# B&R Automation Studio project po_lab4
Automation Studio 4.5.2.102

## Configuration Real

### Hardware
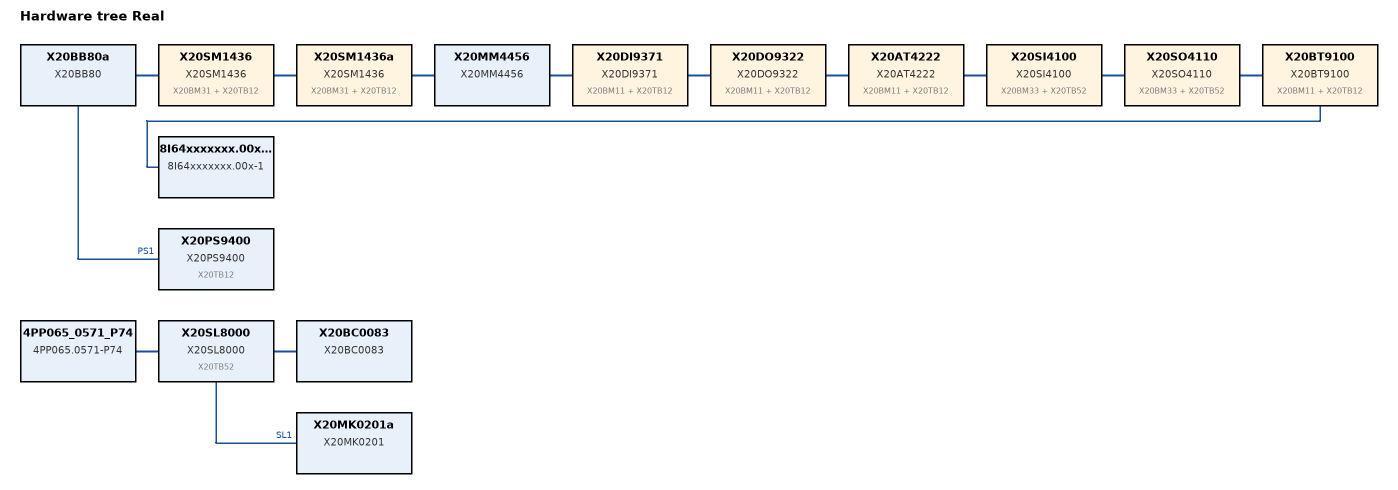
```
4PP065_0571_P74 : 4PP065.0571-P74 v1.1.2.0
  Connector IF4:
    EplInterfaceRedundant = 0
    EplEthInterfaceRedundant = 0
  Connector IF5:
    ActivateDevice = 1
    Mode = Manual
    InternetAddress = 10.0.1.10
    SubnetMask = 255.255.255.0
  ConfigurationID = LabBR
  TimerDeviceType = EPLX2X
  TimerDevice = 4PP065_0571_P74.IF4
  TaskClassIdleTime = 2000
  Cyclic1Tolerance = 0
  Cyclic1Output = 1
  Cyclic3Tolerance = 0
  VcObjectName = Visu
8I64xxxxxxx.00x-1 : 8I64xxxxxxx.00x-1 v1.3.9.1  [X2X1 -> X20BT9100.X2X1 [Cable Type=X2XCable, Length=10, Version=1.0.0.2]]
  BothEndSwitchesAreNormallyOpen_r1 = on
  QuickStopIsNormallyOpen_r1 = on
X20AT4222 : X20AT4222 v1.2.3.0  [SS1 -> X20TB12f.SS; SL -> X20BM11c.SL1]
X20BB80a : X20BB80 v1.0.2.0
X20BC0083 : X20BC0083 v2.7.0.0  [PLK1 -> X20SL8000.PLK2 (NodeNumber=2) [Cable Type=PowerlinkCable, Length=10, Version=1.0.0.2]; SL -> X20BB80a.SL1]
X20BM11a : X20BM11 v1.0.0.1  [X2X1 -> X20MM4456.X2X2]
X20BM11b : X20BM11 v1.0.0.1  [X2X1 -> X20BM11a.X2X2]
X20BM11c : X20BM11 v1.0.0.1  [X2X1 -> X20BM11b.X2X2]
X20BM11d : X20BM11 v1.0.0.1  [X2X1 -> X20BM33b.X2X2]
X20BM31a : X20BM31 v1.0.0.1  [X2X1 -> X20BB80a.IF1]
X20BM31b : X20BM31 v1.0.0.1  [X2X1 -> X20BM31a.X2X2]
X20BM33a : X20BM33 v1.0.0.4  [X2X1 -> X20BM11c.X2X2]
X20BM33b : X20BM33 v1.0.0.4  [X2X1 -> X20BM33a.X2X2]
X20BT9100 : X20BT9100 v1.0.3.0  [SS1 -> X20TB12g.SS; SL -> X20BM11d.SL1]
X20DI9371 : X20DI9371 v1.0.2.0  [SS1 -> X20TB12d.SS; SL -> X20BM11a.SL1]
X20DO9322 : X20DO9322 v1.0.3.0  [SS1 -> X20TB12e.SS; SL -> X20BM11b.SL1]
X20MK0201a : X20MK0201 v1.0.0.0  [SL -> X20SL8000.SL1]
X20MM4456 : X20MM4456 v1.1.5.0  [X2X1 -> X20BM31b.X2X2]
X20PS9400 : X20PS9400 v1.0.2.4  [SS1 -> X20TB12b.SS; PS -> X20BB80a.PS1]
X20SI4100 : X20SI4100 v1.10.1.1  [SS1 -> X20TB52b.SS; SL -> X20BM33a.SL1]
X20SL8000 : X20SL8000 v1.6.5.1  [PLK1 -> 4PP065_0571_P74.IF4 (NodeNumber=1) [Cable Type=PowerlinkCable, Length=10, Version=1.0.0.2]; PLK2 -> X20BC0083.PLK1 (NodeNumber=1) [Cable Type=PowerlinkCable, Length=10, Version=1.0.0.2]; SS1 -> X20TB52a.SS]
  SafeProject = SafeLOGIC-1
X20SM1436 : X20SM1436 v1.4.2.1  [SS1 -> X20TB12a.SS; SL -> X20BM31a.SL1]
X20SM1436a : X20SM1436 v1.4.2.1  [SS1 -> X20TB12c.SS; SL -> X20BM31b.SL1]
X20SO4110 : X20SO4110 v1.10.1.1  [SS1 -> X20TB52c.SS; SL -> X20BM33b.SL1]
  SafeLogicID = 2
  SafeModuleID = 3
X20TB12a : X20TB12 v1.0.0.0
X20TB12b : X20TB12 v1.0.0.0
X20TB12c : X20TB12 v1.0.0.0
X20TB12d : X20TB12 v1.0.0.0
X20TB12e : X20TB12 v1.0.0.0
X20TB12f : X20TB12 v1.0.0.0
X20TB12g : X20TB12 v1.0.0.0
X20TB52a : X20TB52 v1.0.0.1
X20TB52b : X20TB52 v1.0.0.1
X20TB52c : X20TB52 v1.0.0.1
```

### IoMap.iom - 4PP065_0571_P74/IoMap.iom
```iecst
VAR_CONFIG
	::SDCAxisCtr:pwm_period AT %QW."X20MM4456".PeriodDurationPWM;
	::SDCAxisCtr:coil_pwm_value AT %QW."X20MM4456".PulseWidthCurrentPWM04;
	::SDCAxisCtr:axis_X.pwm_value AT %QW."X20MM4456".PulseWidthCurrentPWM01;
	::SDCAxisCtr:axis_X.reset_error AT %QX."X20MM4456".ClearError01;
	::SDCAxisCtr:axis_X.reset_counter AT %QX."X20MM4456".ResetCounter01;
	::AxisX_EncIf.iActPos AT %IW."X20MM4456".Counter01;
	::coil_powered AT %IX."X20DI9371".DigitalInput01;
	::AxisX_DiDoIf.iPosHwEnd AT %IX."X20MM4456".StatusInput03;
	::AxisX_DiDoIf.iNegHwEnd AT %IX."X20MM4456".StatusInput04;
	::SDCAxisCt1:posEnable.enable AT %IX."X20DI9371".DigitalInput02; (*Insert your comment here...*)
	::SDCAxisCt1:posEnableRight.enable AT %IX."X20DI9371".DigitalInput03; (*Insert your comment here...*)
	::SDCAxisCt1:axis_Y.pwm_value AT %QW."X20MM4456".PulseWidthCurrentPWM02;
	::SDCAxisCt2:axis_Z.pwm_value AT %QW."X20MM4456".PulseWidthCurrentPWM03;
	::SDCAxisCt2:axis_Z.reset_counter AT %QX."X20MM4456".ResetCounter03;
	::AxisY_DiDoIf.iPosHwEnd  AT %IX."X20MM4456".StatusInput07;
	::AxisY_DiDoIf.iNegHwEnd  AT %IX."X20MM4456".StatusInput08;
	::AxisZ_DiDoIf.iNegHwEnd  AT %IX."X20MM4456".StatusInput12;
	::AxisZ_DiDoIf.iPosHwEnd  AT %IX."X20MM4456".StatusInput11;
END_VAR
```

### Acp10map.ncm - 4PP065_0571_P74/Motion/Acp10map.ncm
```
NcMapping (NcSwId=ACP10, DisabledNodesAreHidden=False)
  NcObject AxisX (ModuleAddress=SDC_IF1.ST2, InterfaceType=SDC, Type=ncAXIS, Channel=1, AcoposSimulation=Off, InitParameter=gAxis01i, AcoposParameter=gAxis01a, AdditionalData=CNC_Enabled="1" , Disabled=FALSE, ModuleDisabled=FALSE)
  NcObject AxisZ (ModuleAddress=SDC_IF1.ST4, InterfaceType=SDC, Type=ncAXIS, Channel=1, AcoposSimulation=Off, InitParameter=gAxis01i, AcoposParameter=gAxis01a, AdditionalData=CNC_Enabled="1" , Disabled=FALSE)
  NcObject AxisY (ModuleAddress=SDC_IF1.ST3, InterfaceType=SDC, Type=ncAXIS, Channel=1, AcoposSimulation=Off, InitParameter=gAxis01i, AcoposParameter=gAxis01a, AdditionalData=CNC_Enabled="1" , Disabled=FALSE)
```

### Arnc0map.ncm - 4PP065_0571_P74/Motion/Arnc0map.ncm
```
NcMapping (NcSwId=Arnc0, DisabledNodesAreHidden=False)
  NcObject CNC24 (Type=ncCNCSYS, Channel=24, AcoposSimulation=Off, Disabled=TRUE, ModuleDisabled=FALSE)
  NcObject CNC23 (Type=ncCNCSYS, Channel=23, AcoposSimulation=Off, Disabled=TRUE, ModuleDisabled=FALSE)
  NcObject CNC22 (Type=ncCNCSYS, Channel=22, AcoposSimulation=Off, Disabled=TRUE, ModuleDisabled=FALSE)
  NcObject CNC21 (Type=ncCNCSYS, Channel=21, AcoposSimulation=Off, Disabled=TRUE, ModuleDisabled=FALSE)
  NcObject CNC20 (Type=ncCNCSYS, Channel=20, AcoposSimulation=Off, Disabled=TRUE, ModuleDisabled=FALSE)
  NcObject CNC19 (Type=ncCNCSYS, Channel=19, AcoposSimulation=Off, Disabled=TRUE, ModuleDisabled=FALSE)
  NcObject CNC18 (Type=ncCNCSYS, Channel=18, AcoposSimulation=Off, Disabled=TRUE, ModuleDisabled=FALSE)
  NcObject CNC17 (Type=ncCNCSYS, Channel=17, AcoposSimulation=Off, Disabled=TRUE, ModuleDisabled=FALSE)
  NcObject CNC16 (Type=ncCNCSYS, Channel=16, AcoposSimulation=Off, Disabled=TRUE, ModuleDisabled=FALSE)
  NcObject CNC15 (Type=ncCNCSYS, Channel=15, AcoposSimulation=Off, Disabled=TRUE, ModuleDisabled=FALSE)
  NcObject CNC14 (Type=ncCNCSYS, Channel=14, AcoposSimulation=Off, Disabled=TRUE, ModuleDisabled=FALSE)
  NcObject CNC13 (Type=ncCNCSYS, Channel=13, AcoposSimulation=Off, Disabled=TRUE, ModuleDisabled=FALSE)
  NcObject CNC12 (Type=ncCNCSYS, Channel=12, AcoposSimulation=Off, Disabled=TRUE, ModuleDisabled=FALSE)
  NcObject CNC11 (Type=ncCNCSYS, Channel=11, AcoposSimulation=Off, Disabled=TRUE, ModuleDisabled=FALSE)
  NcObject CNC10 (Type=ncCNCSYS, Channel=10, AcoposSimulation=Off, Disabled=TRUE, ModuleDisabled=FALSE)
  NcObject CNC9 (Type=ncCNCSYS, Channel=9, AcoposSimulation=Off, Disabled=TRUE, ModuleDisabled=FALSE)
  NcObject CNC8 (Type=ncCNCSYS, Channel=8, AcoposSimulation=Off, Disabled=TRUE, ModuleDisabled=FALSE)
  NcObject CNC7 (Type=ncCNCSYS, Channel=7, AcoposSimulation=Off, Disabled=TRUE, ModuleDisabled=FALSE)
  NcObject CNC6 (Type=ncCNCSYS, Channel=6, AcoposSimulation=Off, Disabled=TRUE, ModuleDisabled=FALSE)
  NcObject CNC5 (Type=ncCNCSYS, Channel=5, AcoposSimulation=Off, Disabled=TRUE, ModuleDisabled=FALSE)
  NcObject CNC4 (Type=ncCNCSYS, Channel=4, AcoposSimulation=Off, Disabled=TRUE, ModuleDisabled=FALSE)
  NcObject CNC3 (Type=ncCNCSYS, Channel=3, AcoposSimulation=Off, Disabled=TRUE, ModuleDisabled=FALSE)
  NcObject CNC2 (Type=ncCNCSYS, Channel=2, AcoposSimulation=Off, Disabled=TRUE, ModuleDisabled=FALSE)
  NcObject CNCsys (Type=ncCNCSYS, Channel=1, AcoposSimulation=Off, InitParameter=CncInit, AcoposParameter=gAxis01a, Disabled=FALSE, ModuleDisabled=FALSE)
```

## Configuration Simulation

### Task classes (Cpu.sw)
```
Cyclic#1:
  SDCAxisCtr <- SDCAxisCtrl_X.prg
DataObjects: Acp10sys
Binaries: TCData, ashwd, sysconf, asfw, arconfig, iomap, Acp10map, Acp10map1, arnc0cfg, acp10cfg
Libraries: AsIecCon, astime, Acp10sdc, Acp10man, Acp10par, NcGlobal, asstring, AsIOTime, Acp10_MC, brsystem, sys_lib, Runtime, Acp10sim, fileio, powerlnk, Library, AsBrStr
```

## Logical view

### Global.var - Global variables
```iecst
VAR
	coil_powered : BOOL := FALSE;
	AxisX_DrvIf : SdcDrvIf16_typ := (0);
	AxisX_EncIf : SdcEncIf16_typ := (0);
	AxisX_DiDoIf : SdcDiDoIf_typ := (0);
	AxisX_HW : SdcHwCfg_typ := (0);
	AxisY_DrvIf : SdcDrvIf16_typ := (0);
	AxisY_EncIf : SdcEncIf16_typ := (0);
	AxisY_DiDoIf : SdcDiDoIf_typ := (0);
	AxisY_HW : SdcHwCfg_typ := (0);
	AxisZ_DrvIf : SdcDrvIf16_typ := (0);
	AxisZ_EncIf : SdcEncIf16_typ := (0);
	AxisZ_DiDoIf : SdcDiDoIf_typ := (0);
	AxisZ_HW : SdcHwCfg_typ := (0);
	fb_regulator : FB_Regulator;
	iPosHwEnd : BOOL := FALSE;
	iNegHwEnd : BOOL := FALSE;
END_VAR
```

### Package Logical/Libraries - Global libraries

### Library Logical/Libraries/Library (ANSIC)

#### Library.fun
```iecst
FUNCTION_BLOCK FB_Motor (*TODO: Add your comment here*) (*$GROUP=User,$CAT=User,$GROUPICON=User.png,$CATICON=User.png*)
	VAR_INPUT
		in : REAL;
	END_VAR
	VAR_OUTPUT
		out_w : REAL;
		out_phi : REAL;
	END_VAR
	VAR
		k_e : REAL;
		T_m : REAL;
		dt : REAL;
		integrator : FB_Integrator;
		integrator_phi : FB_Integrator;
	END_VAR
END_FUNCTION_BLOCK

FUNCTION_BLOCK FB_Integrator (*TODO: Add your comment here*) (*$GROUP=User,$CAT=User,$GROUPICON=User.png,$CATICON=User.png*)
	VAR_INPUT
		in : REAL;
		dt : REAL;
	END_VAR
	VAR_OUTPUT
		out : REAL;
	END_VAR
	VAR
		state : REAL := 0.0;
	END_VAR
END_FUNCTION_BLOCK

FUNCTION_BLOCK FB_Controller (* *) (*$GROUP=User,$CAT=User,$GROUPICON=User.png,$CATICON=User.png*)
	VAR_INPUT
		in : REAL;
	END_VAR
	VAR_OUTPUT
		out : REAL;
	END_VAR
	VAR
		k_i : REAL;
		sum : REAL;
		k_p : REAL;
		dt : REAL;
		max_abs_value : REAL;
		integrator : FB_Integrator;
		last_sum : REAL;
	END_VAR
END_FUNCTION_BLOCK

FUNCTION_BLOCK FB_Endswitch (*TODO: Add your comment here*) (*$GROUP=User,$CAT=User,$GROUPICON=User.png,$CATICON=User.png*)
	VAR_INPUT
		in : REAL;
		neg_value : REAL;
		pos_value : REAL;
	END_VAR
	VAR_OUTPUT
		neg_reached : BOOL;
		pos_reached : BOOL;
	END_VAR
END_FUNCTION_BLOCK

FUNCTION_BLOCK FB_Axis (*TODO: Add your comment here*) (*$GROUP=User,$CAT=User,$GROUPICON=User.png,$CATICON=User.png*)
	VAR_INPUT
		u : REAL;
		reset_error : BOOL;
		endswitch_a_reached : BOOL;
		endswitch_b_reached : BOOL;
		pwm_percentage : SINT;
	END_VAR
	VAR_OUTPUT
		reset_counter : BOOL;
		pwm_value : INT;
	END_VAR
	VAR_OUTPUT RETAIN
		counter : INT;
	END_VAR
	VAR_OUTPUT
		speed : REAL;
	END_VAR
	VAR
		i : INT;
		last_counter : INT;
		dir : BOOL;
		spid : REAL;
		k : INT;
	END_VAR
END_FUNCTION_BLOCK

{REDUND_ERROR} FUNCTION_BLOCK FB_Regulator (*TODO: Add your comment here*) (*$GROUP=User,$CAT=User,$GROUPICON=User.png,$CATICON=User.png*)
	VAR_INPUT
		e : REAL;
	END_VAR
	VAR_OUTPUT
		u : REAL;
	END_VAR
	VAR
		k_p : REAL;
		k_i : REAL;
		integrator : FB_Integrator;
		iyOld : REAL;
		max_abc_value : REAL := 24;
		dt : REAL;
		x : REAL;
	END_VAR
END_FUNCTION_BLOCK

{REDUND_ERROR} FUNCTION_BLOCK Pos (*TODO: Add your comment here*) (*$GROUP=User,$CAT=User,$GROUPICON=User.png,$CATICON=User.png*)
	VAR_INPUT
		enable : BOOL;
	END_VAR
END_FUNCTION_BLOCK
```

#### FB_Axis.c
```c
#include <bur/plctypes.h>
#ifdef __cplusplus
	extern "C"
	{
#endif
#include "Library.h"
#ifdef __cplusplus
	};
#endif
/* TODO: Add your comment here */
void FB_Axis(struct FB_Axis* inst)
{
	if (inst->endswitch_a_reached == 1 )
	{
		inst->dir = 1;
	}
	if (inst->endswitch_b_reached == 1 )
	{
		inst->dir = 0;
	}

	if(inst->dir == 1)
	{

		//inst->reset_counter = 0;
		inst->u = -inst->u;
		inst->pwm_value = (inst->u/24.0) * 32767;
	}
	if(inst->dir == 0)
	{
		//inst->reset_counter = 0;
		inst->pwm_value = (inst->u/24.0) * 32767;
	}
	if (inst->i == 1000)
	{
		inst->speed = (inst->counter - inst->last_counter)/2;
		inst->last_counter = inst->counter;
		inst->i = 0;
	}
	inst->spid = inst->speed;
	inst->i++;
}
```

#### Pos.c
```c
#include <bur/plctypes.h>
#ifdef __cplusplus
	extern "C"
	{
#endif
	#include "Library.h"
#ifdef __cplusplus
	};
#endif
/* TODO: Add your comment here */
void Pos(struct Pos* inst)
{
	/*TODO: Add your code here*/
}
```

### Package Logical/gAxis01obj - gAxis03obj

### gAxis01a.apt
```
AcoposParameterTable:
  Root Parameters:
    230 = PCTRL_S_SET (Name=PCTRL_S_ACT_PARID)
    64201 = 6500 (Name=SERVO_V_MAX_OUTPUT)
```

### gAxis01i.ax
```
InitParameter (Version=3.13.1, NcSwId=ACP10)
  ACP10AXIS_typ:
    dig_in:
      level:
        reference = ncACTIV_HI
        pos_hw_end = ncACTIV_HI
        neg_hw_end = ncACTIV_HI
        trigger1 = ncACTIV_HI
        trigger2 = ncACTIV_HI
    encoder_if:
      parameter:
        count_dir = ncSTANDARD
        scaling:
          load:
            units = 1000
            rev_motor = 1
    limit:
      parameter:
        v_pos = 10000.0
        v_neg = 10000.0
        a1_pos = 50000.0
        a2_pos = 50000.0
        a1_neg = 50000.0
        a2_neg = 50000.0
        t_jolt = 0.0
        t_in_pos = 0.0
        pos_sw_end = 8388607
        neg_sw_end = -8388608
        ds_warning = 500.0
        ds_stop = 1000.0
        a_stop = 1.0E+30
        dv_stop = 0.0
        dv_stop_mode = ncOFF
    controller:
      mode = ncPOSITION
      position:
        kv = 50.0
        tn = 0.0
        t_predict = 0.01
        t_total = 0.01
        p_max = 1.0E+30
        i_max = 0.0
      speed:
        kv = 2.0
        tn = 0.0
        t_filter = 0.0
        isq_filter1:
          type = ncOFF
          a0 = 0.0
          a1 = 0.0
          b0 = 0.0
          b1 = 0.0
          b2 = 0.0
          c0_par_id = 0
          c1_par_id = 0
        isq_filter2:
          type = ncOFF
          a0 = 0.0
          a1 = 0.0
          b0 = 0.0
          b1 = 0.0
          b2 = 0.0
          c0_par_id = 0
          c1_par_id = 0
        isq_filter3:
          type = ncOFF
          a0 = 0.0
          a1 = 0.0
          b0 = 0.0
          b1 = 0.0
          b2 = 0.0
          c0_par_id = 0
          c1_par_id = 0
      uf:
        type = ncLINEAR
        auto_config = ncMOTOR_PAR
        u0 = 0.0
        un = 0.0
        fn = 50.0
        k_f_slip = 0.0
      ff:
        torque_load = 0.0
        torque_pos = 0.0
        torque_neg = 0.0
        kv_torque = 0.0
        inertia = 0.0
        t_filter_a = 0.0
    move:
      stop:
        parameter[0]:
          decel_ramp = ncA_LIMIT
          controller = ncON
        parameter[1]:
          decel_ramp = ncA_LIMIT
          controller = ncON
        parameter[2]:
          decel_ramp = ncA_LIMIT
          controller = ncON
        parameter[3]:
          decel_ramp = ncA_LIMIT
          controller = ncON
        quickstop:
          decel_ramp = ncA_LIMIT
        drive_error:
          decel_ramp = ncA_LIMIT
      homing:
        parameter:
          s = 0
          v_switch = 5000.0
          v_trigger = 500.0
          a = 50000.0
          mode = ncEND_SWITCH
          edge_sw = ncPOSITIVE
          start_dir = ncPOSITIVE
          trigg_dir = ncPOSITIVE
          ref_pulse = ncOFF
          fix_dir = ncOFF
          tr_s_block = 0.0
          torque_lim = 0.0
          ds_block = 0.0
          ds_stop = 0.0
      basis:
        parameter:
          v_pos = 5000.0
          v_neg = 5000.0
          a1_pos = 50000.0
          a2_pos = 50000.0
          a1_neg = 50000.0
          a2_neg = 50000.0
    message:
      text:
        parameter:
          format = ncBREAK
          columns = 80
          data_modul = acp10etxen
```

### Program Logical/SDCAxisCtrl_X (ANSIC)

#### Variables.var
```iecst
VAR
	axis_X : FB_Axis;
	coil_pwm_value : {REDUND_UNREPLICABLE} INT := 200;
	pwm_period : {REDUND_UNREPLICABLE} UINT := 200;
	Already_Homed : BOOL := FALSE;
	k : INT := 0;
	posEnable : Pos := (0);
	posEnableRight : Pos := (0);
END_VAR
```

#### Main.c
```c
#include <bur/plctypes.h>

#ifdef _DEFAULT_INCLUDES
#include <AsDefault.h>
#endif

void increase_counters(void);
void Homing(void);

void _INIT ProgramInit(void)
{
	AxisX_HW.EncIf1_Typ = ncSDC_ENC16;
	AxisX_HW.DiDoIf_Typ = ncSDC_DIDO;
	AxisX_HW.DrvIf_Typ  = ncSDC_DRVSERVO16;

	strcpy(AxisX_HW.EncIf1_Name, "AxisX_EncIf");
	strcpy(AxisX_HW.DrvIf_Name,   "AxisX_DrvIf");
	strcpy(AxisX_HW.DiDoIf_Name,  "AxisX_DiDoIf");

	AxisX_EncIf.iEncOK        = 1;
	AxisX_DrvIf.iDrvOK        = 1;
	AxisX_DrvIf.iStatusEnable = 1;
	AxisX_DiDoIf.iDriveReady  = 1;

	fb_regulator.dt            = 0.002;
	fb_regulator.k_i           = 0.16;
	fb_regulator.k_p           = 0.0064;
	fb_regulator.max_abc_value = 24.0;

	pwm_period = 200;
}

void _CYCLIC ProgramCyclic(void)
{
	if (posEnable.enable)
	{
		AxisX_DrvIf.oSetPos = -10000;
	}
	else if (posEnableRight.enable)
	{
		AxisX_DrvIf.oSetPos = 10000;
	}

	increase_counters();
	AxisX_EncIf.iActTime = (INT)AsIOTimeCyclicStart();

	AxisX_DiDoIf.iPosHwEnd = axis_X.endswitch_a_reached;
	AxisX_DiDoIf.iNegHwEnd = axis_X.endswitch_b_reached;

	if (coil_powered == 0)
	{
		coil_pwm_value = 0;

		fb_regulator.e = 0;
		FB_Regulator(&fb_regulator);

		axis_X.u = 0;
		FB_Axis(&axis_X);
	}
	else
	{
			increase_counters();

			axis_X.reset_counter = 0;
			FB_Axis(&axis_X);

			coil_pwm_value = 32767;

			iPosHwEnd = axis_X.endswitch_a_reached;
			iNegHwEnd = axis_X.endswitch_b_reached;
			FB_Axis(&axis_X);

			fb_regulator.e = (AxisX_DrvIf.oSetPos * 10) - axis_X.speed;
			FB_Regulator(&fb_regulator);

			axis_X.u = fb_regulator.u;
			FB_Axis(&axis_X);
	}

}

void increase_counters(void)
{
	AxisX_EncIf.iLifeCnt++;

	AxisX_DiDoIf.iLifeCntDriveEnable++;
	AxisX_DiDoIf.iLifeCntDriveReady++;
	AxisX_DiDoIf.iLifeCntNegHwEnd++;
	AxisX_DiDoIf.iLifeCntPosHwEnd++;
	AxisX_DiDoIf.iLifeCntReference++;

	AxisX_DrvIf.iLifeCnt++;
}

void _EXIT ProgramExit(void)
{
}
```

### Program Logical/SDCAxisCtrl_Y (ANSIC)

#### Variables.var
```iecst
VAR
	axis_Y : FB_Axis;
	coil_pwm_value : {REDUND_UNREPLICABLE} INT := 200;
	pwm_period : {REDUND_UNREPLICABLE} UINT := 200;
	Already_Homed : BOOL := FALSE;
	k : INT := 0;
	posEnable : Pos := (0);
	posEnableRight : Pos := (0);
END_VAR
```

#### Main.c
```c
#include <bur/plctypes.h>

#ifdef _DEFAULT_INCLUDES
#include <AsDefault.h>
#endif

void increase_counters(void);
void Homing(void);

void _INIT ProgramInit(void)
{
	AxisY_HW.EncIf1_Typ = ncSDC_ENC16;
	AxisY_HW.DiDoIf_Typ = ncSDC_DIDO;
	AxisY_HW.DrvIf_Typ  = ncSDC_DRVSERVO16;

	strcpy(AxisY_HW.EncIf1_Name, "AxisY_EncIf");
	strcpy(AxisY_HW.DrvIf_Name,   "AxisY_DrvIf");
	strcpy(AxisY_HW.DiDoIf_Name,  "AxisY_DiDoIf");

	AxisY_EncIf.iEncOK        = 1;
	AxisY_DrvIf.iDrvOK        = 1;
	AxisY_DrvIf.iStatusEnable = 1;
	AxisY_DiDoIf.iDriveReady  = 1;

	fb_regulator.dt            = 0.002;
	fb_regulator.k_i           = 0.16;
	fb_regulator.k_p           = 0.0064;
	fb_regulator.max_abc_value = 24.0;

	pwm_period = 200;
}

void _CYCLIC ProgramCyclic(void)
{
	if (posEnable.enable)
	{
		AxisY_DrvIf.oSetPos = -10000;
	}
	else if (posEnableRight.enable)
	{
		AxisY_DrvIf.oSetPos = 10000;
	}

	increase_counters();
	AxisY_EncIf.iActTime = (INT)AsIOTimeCyclicStart();

	AxisY_DiDoIf.iPosHwEnd = axis_Y.endswitch_a_reached;
	AxisY_DiDoIf.iNegHwEnd = axis_Y.endswitch_b_reached;

	if (coil_powered == 0)
	{
		coil_pwm_value = 0;

		fb_regulator.e = 0;
		FB_Regulator(&fb_regulator);

		axis_Y.u = 0;
		FB_Axis(&axis_Y);
	}
	else
	{
			increase_counters();

			axis_Y.reset_counter = 0;
			FB_Axis(&axis_Y);

			coil_pwm_value = 32767;

			iPosHwEnd = axis_Y.endswitch_a_reached;
			iNegHwEnd = axis_Y.endswitch_b_reached;
			FB_Axis(&axis_Y);

			fb_regulator.e = (AxisY_DrvIf.oSetPos * 10) - axis_Y.speed;
			FB_Regulator(&fb_regulator);

			axis_Y.u = fb_regulator.u;
			FB_Axis(&axis_Y);
	}

}

void increase_counters(void)
{
	AxisY_EncIf.iLifeCnt++;

	AxisY_DiDoIf.iLifeCntDriveEnable++;
	AxisY_DiDoIf.iLifeCntDriveReady++;
	AxisY_DiDoIf.iLifeCntNegHwEnd++;
	AxisY_DiDoIf.iLifeCntPosHwEnd++;
	AxisY_DiDoIf.iLifeCntReference++;

	AxisY_DrvIf.iLifeCnt++;
}

void _EXIT ProgramExit(void)
{
}
```

### Program Logical/SDCAxisCtrl_Z (ANSIC)

#### Variables.var
```iecst
VAR
	axis_Z : FB_Axis;
	coil_pwm_value : {REDUND_UNREPLICABLE} INT := 200;
	pwm_period : {REDUND_UNREPLICABLE} UINT := 200;
	Already_Homed : BOOL := FALSE;
	k : INT := 0;
	posEnable : Pos := (0);
	posEnableRight : Pos := (0);
END_VAR
```

#### Main.c
```c
#include <bur/plctypes.h>

#ifdef _DEFAULT_INCLUDES
#include <AsDefault.h>
#endif

void increase_counters(void);
void Homing(void);

void _INIT ProgramInit(void)
{
	AxisZ_HW.EncIf1_Typ = ncSDC_ENC16;
	AxisZ_HW.DiDoIf_Typ = ncSDC_DIDO;
	AxisZ_HW.DrvIf_Typ  = ncSDC_DRVSERVO16;

	strcpy(AxisZ_HW.EncIf1_Name, "AxisZ_EncIf");
	strcpy(AxisZ_HW.DrvIf_Name,   "AxisZ_DrvIf");
	strcpy(AxisZ_HW.DiDoIf_Name,  "AxisZ_DiDoIf");

	AxisZ_EncIf.iEncOK        = 1;
	AxisZ_DrvIf.iDrvOK        = 1;
	AxisZ_DrvIf.iStatusEnable = 1;
	AxisZ_DiDoIf.iDriveReady  = 1;

	fb_regulator.dt            = 0.002;
	fb_regulator.k_i           = 0.16;
	fb_regulator.k_p           = 0.0064;
	fb_regulator.max_abc_value = 24.0;

	pwm_period = 200;
}

void _CYCLIC ProgramCyclic(void)
{
	if (posEnable.enable)
	{
		AxisZ_DrvIf.oSetPos = -10000;
	}
	else if (posEnableRight.enable)
	{
		AxisZ_DrvIf.oSetPos = 10000;
	}

	increase_counters();
	AxisZ_EncIf.iActTime = (INT)AsIOTimeCyclicStart();

	AxisZ_DiDoIf.iPosHwEnd = axis_Z.endswitch_a_reached;
	AxisZ_DiDoIf.iNegHwEnd = axis_Z.endswitch_b_reached;

	if (coil_powered == 0)
	{
		coil_pwm_value = 0;

		fb_regulator.e = 0;
		FB_Regulator(&fb_regulator);

		axis_Z.u = 0;
		FB_Axis(&axis_Z);
	}
	else
	{
			increase_counters();

			axis_Z.reset_counter = 0;
			FB_Axis(&axis_Z);

			coil_pwm_value = 32767;

			iPosHwEnd = axis_Z.endswitch_a_reached;
			iNegHwEnd = axis_Z.endswitch_b_reached;
			FB_Axis(&axis_Z);

			fb_regulator.e = (AxisZ_DrvIf.oSetPos * 10) - axis_Z.speed;
			FB_Regulator(&fb_regulator);

			axis_Z.u = fb_regulator.u;
			FB_Axis(&axis_Z);
	}

}

void increase_counters(void)
{
	AxisZ_EncIf.iLifeCnt++;

	AxisZ_DiDoIf.iLifeCntDriveEnable++;
	AxisZ_DiDoIf.iLifeCntDriveReady++;
	AxisZ_DiDoIf.iLifeCntNegHwEnd++;
	AxisZ_DiDoIf.iLifeCntPosHwEnd++;
	AxisZ_DiDoIf.iLifeCntReference++;

	AxisZ_DrvIf.iLifeCnt++;
}

void _EXIT ProgramExit(void)
{
}
```

### Data object Logical/CncInit (Cns)

- CncInit.cns (not shown)

### Data object Logical/CncProg (Cnc)

#### CncProg.cnc
```
%001 (CncProgram)

N10 G01 X0 Y-30000 Z0 F300000
N11 G01 X0 Y0 Z-30000  F300000

N999 M30
```

- Data object Logical/GmcIpUserConfig/gmcipvar (Cnc, version 3.13.0) (no source held here)

- Data object Logical/GmcIpUserConfig/gmcipfun (Cnc, version 3.13.0) (no source held here)

- Data object Logical/GmcIpUserConfig/gmcipfub (Cnc, version 3.13.0) (no source held here)

- Data object Logical/GmcIpUserConfig/gmcipubr (Cnc, version 3.13.0) (no source held here)

- Data object Logical/GmcIpUserConfig/gmcipusm (Cnc, version 3.13.0) (no source held here)

- Data object Logical/GmcIpUserConfig/gmcipui (Cnc, version 3.13.0) (no source held here)

- Data object Logical/GmcIpUserConfig/gmcipus (Cnc, version 3.13.0) (no source held here)

- Data object Logical/GmcIpUserConfig/gmcipuc (Cnc, version 3.13.0) (no source held here)

- Data object Logical/GmcIpConfig/gmcipsys (Cnc, version 3.13.0) (no source held here)

- Data object Logical/GmcIpConfig/gmciplbr (Cnc, version 3.13.0) (no source held here)

- Data object Logical/GmcIpConfig/gmcipcbr (Cnc, version 3.13.0) (no source held here)

- Data object Logical/GmcIpConfig/gmciplsm (Cnc, version 3.13.0) (no source held here)

- Data object Logical/GmcIpConfig/gmcipcsm (Cnc, version 3.13.0) (no source held here)

- Data object Logical/GmcIpConfig/gmcipcfg (Cnc, version 3.13.0) (no source held here)

- Data object Logical/GmcIpConfig/gmcipiec (Cnc, version 3.13.0) (no source held here)

- Data object Logical/GmcIpConfig/gmciplog (Cnc, version 3.13.0) (no source held here)

- Data object Logical/GmcIpConfig/gmcipesm (Cnc, version 3.13.0) (no source held here)

- Data object Logical/GmcIpConfig/gmcipmxd (Cnc, version 3.13.0) (no source held here)

- Data object Logical/GmcIpConfig/gmcipmx (Cnc, version 3.13.0) (no source held here)

Listed in the project but not available here: Logical/Global.typ, Logical/Libraries/Library/FB_Motor.c, Logical/Libraries/Library/FB_Controller.c, Logical/Libraries/Library/FB_Integrator.c, Logical/Libraries/Library/FB_Endswitch.c, Logical/Libraries/Library/FB_Regulator.c, Logical/Types.typ
